FUNCTION_BLOCK Fb_RealToAnalog_Conversion
VAR_INPUT
	lActualVal	: REAL;
	lMinVal		: REAL;
	lMaxVal		: REAL;
	
END_VAR
VAR_OUTPUT
	iRawVal	: UINT;					//Raw converted sensor values
END_VAR           
VAR               
	lRangeHigh	: REAL := 32676;
	lRawVal : REAL;

END_VAR


IF lActualVal <=0 THEN
	iRawVal:=0;
END_IF

IF lActualVal>0 THEN
	lRawVal:=(lActualVal-lMinVal)*((lRangeHigh-0)/(lMaxVal-lMinVal));
END_IF

END_FUNCTION_BLOCK

(* stored: Version 1.1.0.1, ProductVersion 3.1.4024.12
   POU Fb_RealToAnalog_Conversion: Id {155a943d-b153-4106-9f22-5ea1cec92c87}, SpecialFunc None *)
